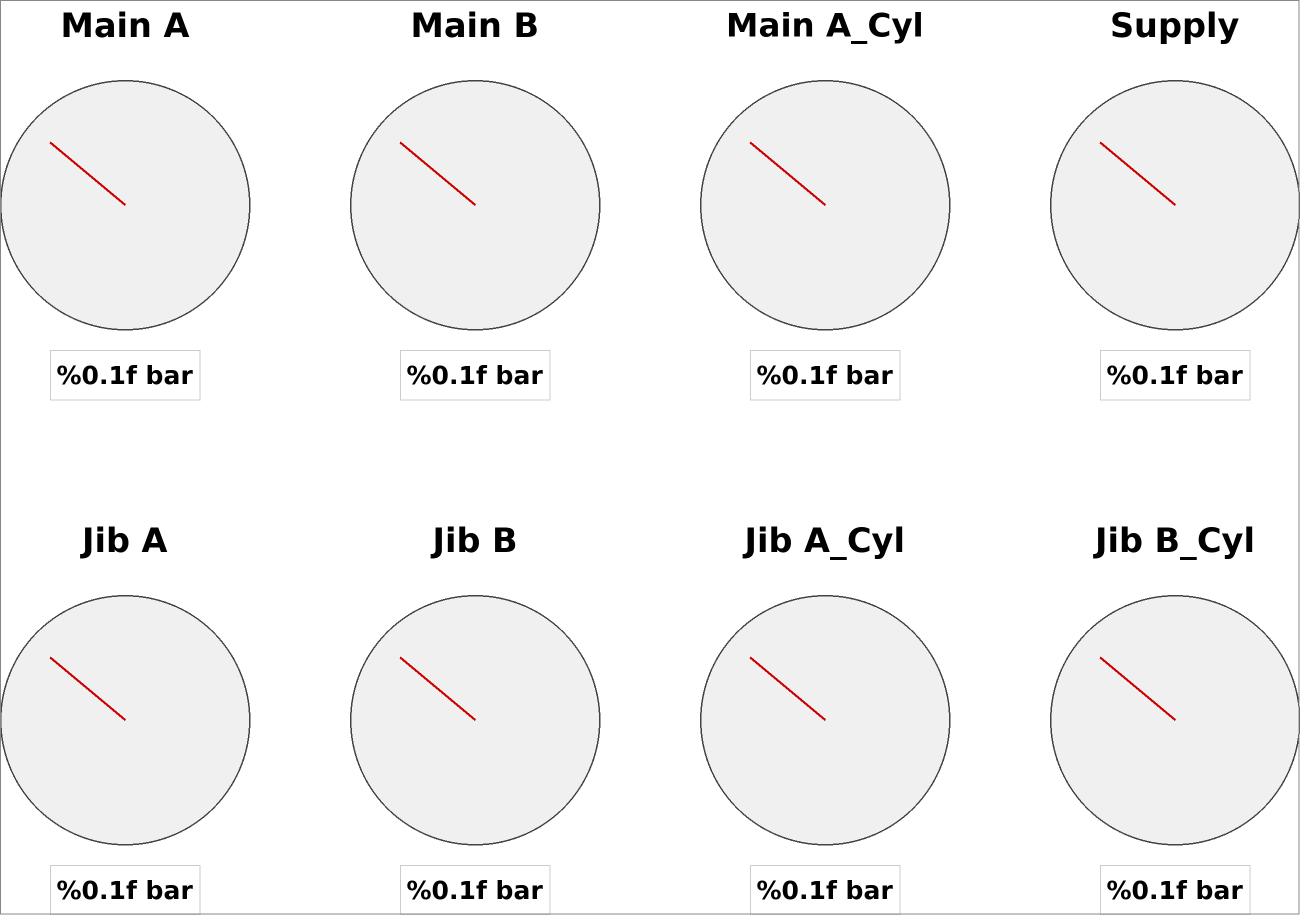
VISUALIZATION VISU_Pressure  // 1300x915
    Textfield (50,0 150x50), "Main A"
    Textfield (375,0 200x50), "Main B"
    Meter360 (350,80 250x250), value: fMain_Pb_bar, style: Meter-Meter360-Gray, scale format: %.1f, scale 0..250
    Meter360 (700,80 250x250), value: fMain_Pa_Cyl_bar, style: Meter-Meter360-Gray, scale format: %.1f, scale 0..250
    Textfield (725,0 200x50), "Main A_Cyl"
    Meter360 (0,80 250x250), value: fMain_Pa_bar, style: Meter-Meter360-Gray, scale format: %.1f, scale 0..250
    Meter360 (1050,80 250x250), value: fPs_bar, style: Meter-Meter360-Gray, scale format: %.1f, scale 0..250
    Textfield (1075,0 200x50), "Supply"
    Textfield (50,350 150x50), "%0.1f bar", text variable: fMain_Pa_bar
    Textfield (400,350 150x50), "%0.1f bar", text variable: fMain_Pb_bar
    Textfield (750,350 150x50), "%0.1f bar", text variable: fMain_Pa_Cyl_bar
    Textfield (1100,350 150x50), "%0.1f bar", text variable: fPs_bar
    Textfield (50,515 150x50), "Jib A"
    Textfield (725,515 200x50), "Jib A_Cyl"
    Meter360 (700,595 250x250), value: fJib_Pa_Cyl_bar, style: Meter-Meter360-Gray, scale format: %.1f, scale 0..250
    Meter360 (350,595 250x250), value: fJib_Pb_bar, style: Meter-Meter360-Gray, scale format: %.1f, scale 0..250
    Textfield (375,515 200x50), "Jib B"
    Meter360 (0,595 250x250), value: fJib_Pa_bar, style: Meter-Meter360-Gray, scale format: %.1f, scale 0..250
    Meter360 (1050,595 250x250), value: fJib_Pb_Cyl_bar, style: Meter-Meter360-Gray, scale format: %.1f, scale 0..250
    Textfield (1075,515 200x50), "Jib B_Cyl"
    Textfield (50,865 150x50), "%0.1f bar", text variable: fJib_Pa_bar
    Textfield (750,865 150x50), "%0.1f bar", text variable: fJib_Pa_Cyl_bar
    Textfield (400,865 150x50), "%0.1f bar", text variable: fJib_Pb_bar
    Textfield (1100,865 150x50), "%0.1f bar", text variable: fJib_Pb_Cyl_bar
END_VISUALIZATION

(* stored: Version 1.1.0.1
   Visu VISU_Pressure: Id {5ea15039-a163-4a3a-90d4-4bb2d35557f0} *)
